FUNCTION_BLOCK Conveyor 
VAR_INPUT
END_VAR

VAR_OUTPUT
	bStart  : BOOL;
END_VAR
VAR
	fbStart : BoolOut;
END_VAR

bStart := fbStart.getValue;

PROPERTY getStart : BoolOut
GET
getStart := fbStart;
END_GET
END_PROPERTY

METHOD Off : BOOL
VAR_INPUT
END_VAR
END_METHOD

METHOD On : BOOL
VAR_INPUT
END_VAR
END_METHOD

END_FUNCTION_BLOCK

(* stored: Version 1.1.0.1, ProductVersion 3.1.4024.0
   POU Conveyor: Id {b15311d8-a9f4-4077-9cec-ef51ff0c9999}, SpecialFunc None
   Property getStart: Id {6370b0c0-d40e-456d-89ce-6f31c418ed60}
   Get Get: Id {489b8359-b98c-42ae-afe2-3461bd22238e}
   Method Off: Id {f085c888-d730-4182-bd45-298546b54d73}
   Method On: Id {5d342f49-f715-42fd-b4a3-ca7fc5d5e1e7} *)
